TYPE ST_PLC_events :
STRUCT
	b_EthercatMasterFault		: BOOL;
END_STRUCT
END_TYPE

(* stored: Version 1.1.0.1, ProductVersion 3.1.4026.18
   DUT ST_PLC_events: Id {2394b53c-8fd9-42d4-9733-0aef698c16d3} *)
